TYPE T_RejectCode : STRING[100];
END_TYPE

(* stored: Version 1.1.0.1
   DUT T_RejectCode: Id {42474b9a-9861-43e9-8e01-2686423af164} *)
